Staubli VAL3: saveFile.pgx

public program saveFile(num x_nCamID (dimensions=1), string x_sJob (dimensions=1), bool& x_bError[] (dimensions=1))
begin
  //-----------------------------------------------------------------------
  //Header begin
  //Description of program
  //  Saves the current job in flash memory on the In-Sight sensor
  //  attached to camera's ID.
  //
  //!!! The In-Sight sensor must be Offline  !!!
  //Input parameters
  //  num x_nCamID :
  //    role : camera's ID
  //  string x_sJob :
  //    role : The name of the job. The file extension must be .JOB.
  //
  //Output parameters
  //  bool x_bError :
  //    role : returns true if an error occurred and false otherwise
  //
  //Examples
  //  call saveFile(nCamID,"example.job",l_bError)
  //
  //History
  //  Creation : 19-05-08 - f.Rob
  //Header end
  //-----------------------------------------------------------------------

  nProgram[x_nCamID]=6
  call sendCommand(x_nCamID,"TF"+x_sJob,x_bError)
end
